INTERFACE IFileHandleTask EXTENDS IFileSystemTask

{attribute 'monitoring' := 'call'}
PROPERTY FileHandle : UINT
GET
END_GET
END_PROPERTY

{attribute 'monitoring' := 'call'}
PROPERTY FINAL FilePath : Tc2_System.T_MaxString
GET
END_GET
END_PROPERTY

METHOD SetFileOpen
VAR_INPUT
	fileOpen : REFERENCE TO Tc2_System.FB_FileOpen;
END_VAR
END_METHOD

END_INTERFACE

(* stored: Version 1.1.0.1
   Itf IFileHandleTask: Id {859cad29-f756-4643-9494-4f576dede29b}
   Property FileHandle: Id {f6c6e0fd-429b-4e98-bf0d-619a28a96627}
   Get Get: Id {83d0effd-8aa4-4f4d-b6d8-9e5a583ecb21}
   Property FilePath: Id {60cfe4a8-0551-4d90-aecd-e47e23f80131}
   Get Get: Id {c6b874d6-1ea7-49dc-9993-89439dc6a142}
   Method SetFileOpen: Id {4580e1bd-b58f-4c03-b06a-eb0706e8e9f9} *)
